TYPE TYP_HW_L4000_EXT_CTRL :
STRUCT
	Trigger AT %Q* : ARRAY[0..7] OF BOOL;
END_STRUCT
END_TYPE

(* stored: Version 1.1.0.1, ProductVersion 3.1.4024.12
   DUT TYP_HW_L4000_EXT_CTRL: Id {9ff255ba-b944-4ef3-8a53-bb31267591c4} *)
